// TIA Portal project "LAB5" (V18)

(* hardware
DEVICE "S7-1500/ET200MP station_1"  S7-1500 station
   slot 0: "Rail_0"  Rack  6ES7 590-1***0-0AA0
   slot 1: "PLC_1"  CPU 1511-1 PN  6ES7 511-1AK00-0AB0  V1.8
      slot 3: "CPU display_1"  6ES7591-1AA00-0AA0
      slot 32768: "PROFINET interface_1"  X1
         slot 32769: "Port_1"  X1 P1
         slot 32770: "Port_2"  X1 P2
   slot 2: "CM 1542-5_1"  CM 1542-5  6GK7 542-5DX00-0XE0  V1.0
   slot 3: "DI 16x24VDC HF_1"  DI 16x24VDC HF  6ES7 521-1BH00-0AB0  V2.0
   slot 4: "DQ 16x24VDC/0.5A ST_1"  DQ 16x24VDC/0.5A ST  6ES7 522-1BH00-0AB0  V2.0
   slot 5: "AI 8xU/I/RTD/TC ST_1"  AI 8xU/I/RTD/TC ST  6ES7 531-7KF00-0AB0  V1.0
   slot 6: "AQ 4xU/I ST_1"  AQ 4xU/I ST  6ES7 532-5HD00-0AB0  V1.0
DEVICE "GSD device_1"  GSD.Device
   slot 0: "Rack_0"  Rail
   slot 0: "Slave_1"  6SE640X-1PB00-0AA0  V1.0
DEVICE "HMI_1"  KTP600 Basic color PN
   slot 0: "HMI_1"  KTP600 Basic color PN  6AV6 647-0AD11-3AX0  12.0.0.0
   slot 1: "HMI_RT_1"  KTP600 Basic color PN  6AV6 647-0AD11-3AX0  12.0.0.0
   slot 5: "HMI_1.IE_CP_1"  PROFINET Interface  12.0.0.0
      slot 1: "PROFINET Interface_1"  PROFINET Interface
         slot 1: "Port_1"  Port
DEVICE "PC-System_1"  SIMATIC PC station
   slot 0: "SIMATIC PC station"  Rail  SIMATIC PC-Station  V1.0
      slot 125: "Stationmanager"  Station_Manager  V6.0.4
   slot 1: "HMI_RT_2"  WinCC RT Advanced  6AV2 104-0xxxx-xxxx  16.0.0.0
      slot 33792: "Computer interface"  Host interface
   slot 2: "IE general_1"  IE General  IE_CP  V8.2.0
      slot 1: "PROFINET interface"  IEGeneral.Interface.8.2.0
*)

// ===== PLC "PLC_1"  CPU 1511-1 PN =====

VAR_GLOBAL   // PLC tag table "Default tag table"
   "inicio_variador" AT %M0.0 : Bool;
   "Tag_19" AT %M0.1 : Bool;
   "Tag_20" AT %M0.2 : Bool;
   "Tag_21" AT %M0.3 : Bool;
   "Tag_22" AT %M0.4 : Bool;
   "Tag_23" AT %M0.5 : Bool;
   "Tag_24" AT %M0.6 : Bool;
   "Tag_25" AT %M0.7 : Bool;
   "Tag_26" AT %M1.0 : Bool;
   "Tag_27" AT %M1.1 : Bool;
   "Tag_28" AT %M1.2 : Bool;
   "Tag_29" AT %M1.3 : Bool;
   "Tag_30" AT %M1.4 : Bool;
   "Tag_31" AT %M1.5 : Bool;
   "Tag_32" AT %M1.6 : Bool;
   "Tag_33" AT %M1.7 : Bool;
   "Tag_34" AT %M2.0 : Bool;
   "Tag_1" AT %ID18 : DWord;
   "Palabramando" AT %QW18 : Word;
   "velocidadescribir" AT %QW20 : Int;
   "Tag_2" AT %MW90 : Int;
   "palabraestado" AT %IW26 : Word;
   "parametro" AT %QW10 : Word;
   "indice" AT %QW12 : Word;
   "valorparametro" AT %QD14 : DWord;
   "Tag_4" AT %QW16 : Word;
   "leerparametro" AT %IW18 : Word;
   "paramrecib" AT %MW4 : Word;
   "indicerecib" AT %MW6 : Word;
   "leerindice" AT %IW20 : Word;
   "leervalparametro" AT %ID22 : DWord;
   "valorparamrecib" AT %MD8 : DWord;
   "aux_SP" AT %IW12 : Int;
   "SP" AT %MD16 : Real;
   "Visual_SP" AT %QW22 : Int;
   "aux_Sensor" AT %IW24 : Int;
   "Level_Sensor" AT %MD28 : Real;
   "Visual_Sensor" AT %QW32 : Int;
   "Q_PID" AT %MD36 : Real;
   "Error" AT %MD62 : Real;
   "Start" AT %I0.0 : Bool;
   "Stop" AT %M48.1 : Bool;
   "Emergency" AT %M48.2 : Bool;
   "ON/OFF" AT %M48.3 : Bool;
   "PID" AT %M48.4 : Bool;
   "END" AT %M48.5 : Bool;
   "Reset" AT %M48.6 : Bool;
   "M_Level_CM" AT %MD49 : Real;
   "HMI_SP" AT %MD53 : Real;
   "Q_VFD_Speed" AT %MW58 : Int;
   "Q_Indc_Alarm" AT %Q60.1 : Bool;
   "Q_Indc_Start" AT %Q60.2 : Bool;
   "Q_Indc_Stop" AT %Q60.3 : Bool;
   "Clock1.5Hz" AT %Q60.4 : Bool;
   "Q_Valve" AT %Q60.5 : Bool;
   "M_Limit_Histerisis" AT %QD61 : Real;
   "On_factory" AT %M66.0 : Bool;
   "On_Analogic" AT %M66.1 : Bool;
   "L_Level_Raw" AT %MW67 : Int;
   "L_Level_m" AT %MD70 : Real;
   "SP_%" AT %MD74 : Real;
   "Sensor_%" AT %MD78 : Real;
   "SP_cm" AT %MD82 : Real;
   "Sensor_cm" AT %MD86 : Real;
   "Q_PID_aux" AT %MD92 : Real;
   "M_PID" AT %MD96 : Real;
   "Q_factory" AT %MW120 : Int;
   "Filling" AT %MW102 : Int;
   "Emptying" AT %MW104 : Int;
   "In_Pot" AT %ID30 : Real;
   "In_Sensor" AT %ID34 : Real;
   "Q_PUMP1" AT %QD30 : Real;
   "Q_PUMP2" AT %QD34 : Real;
END_VAR

TYPE "inn"
   STRUCT
      Mandoderecha : Bool;
      Mandoizquierdo : Bool;
      ControldesdePLC : Bool;
      Inversionvalorconsigna : Bool;
      Noutilizado : Bool;
      Potenciometrohaciaarriba : Bool;
      Potenciometrohaciaabajo : Bool;
      "Local/remoto" : Bool;
      "ON/OFF1" : Bool;
      OFF2stopelectrico : Bool;
      OFF3stoprapido : Bool;
      Activarpulsos : Bool;
      Activargeneradorrampa : Bool;
      Generadorrampa : Bool;
      Activarvalorconsigna : Bool;
      Acusedefallo : Bool;
      Velocidadvariador : Int;
   END_STRUCT;
END_TYPE

TYPE "out"
   STRUCT
      Sindesviacionvalreaconsigna : Bool;
      Controlsolicitado : Bool;
      frecuenciasalida : Bool;
      alarma : Bool;
      freno : Bool;
      sobrecarga : Bool;
      giro : Bool;
      sobrecargaconvertidor : Bool;
      listoparaservicio : Bool;
      listoparaarrancar : Bool;
      serviciodesbloqueado : Bool;
      fallo : Bool;
      "comando aus2/off2" : Bool;
      "comandoaus3/off3" : Bool;
      Bloqueodearranque : Bool;
      Alarmas : Bool;
      Velocidadactual : Int;
   END_STRUCT;
END_TYPE

DATA_BLOCK "lect_variador"   // DB1
{ S7_Optimized_Access := 'FALSE' }
VERSION : 0.1
   VAR
      estadovariador : "out";
   END_VAR
BEGIN
END_DATA_BLOCK

DATA_BLOCK "esc_variador"   // DB2
{ S7_Optimized_Access := 'FALSE' }
VERSION : 0.1
   VAR
      esc_variador : "inn";
   END_VAR
BEGIN
END_DATA_BLOCK

DATA_BLOCK "Variator_DB"   // DB3
{ S7_Optimized_Access := 'TRUE' }
VERSION : 0.1
// stored: InstanceOfName Variator
"Variator"
BEGIN
END_DATA_BLOCK

DATA_BLOCK "SETPOINT_DB"   // DB5
{ S7_Optimized_Access := 'TRUE' }
VERSION : 0.1
// stored: InstanceOfName SETPOINT
"SETPOINT"
BEGIN
END_DATA_BLOCK

DATA_BLOCK "SENSOR_DB"   // DB6
{ S7_Optimized_Access := 'TRUE' }
VERSION : 0.1
// stored: InstanceOfName SENSOR
"SENSOR"
BEGIN
END_DATA_BLOCK

DATA_BLOCK "OUT_PID_DB"   // DB7
{ S7_Optimized_Access := 'TRUE' }
VERSION : 0.1
// stored: InstanceOfName OUT_PID
"OUT_PID"
BEGIN
END_DATA_BLOCK

FUNCTION_BLOCK "Variator"   // FB1, LAD
{ S7_Optimized_Access := 'TRUE' }
VERSION : 0.1
BEGIN

REGION Network 1
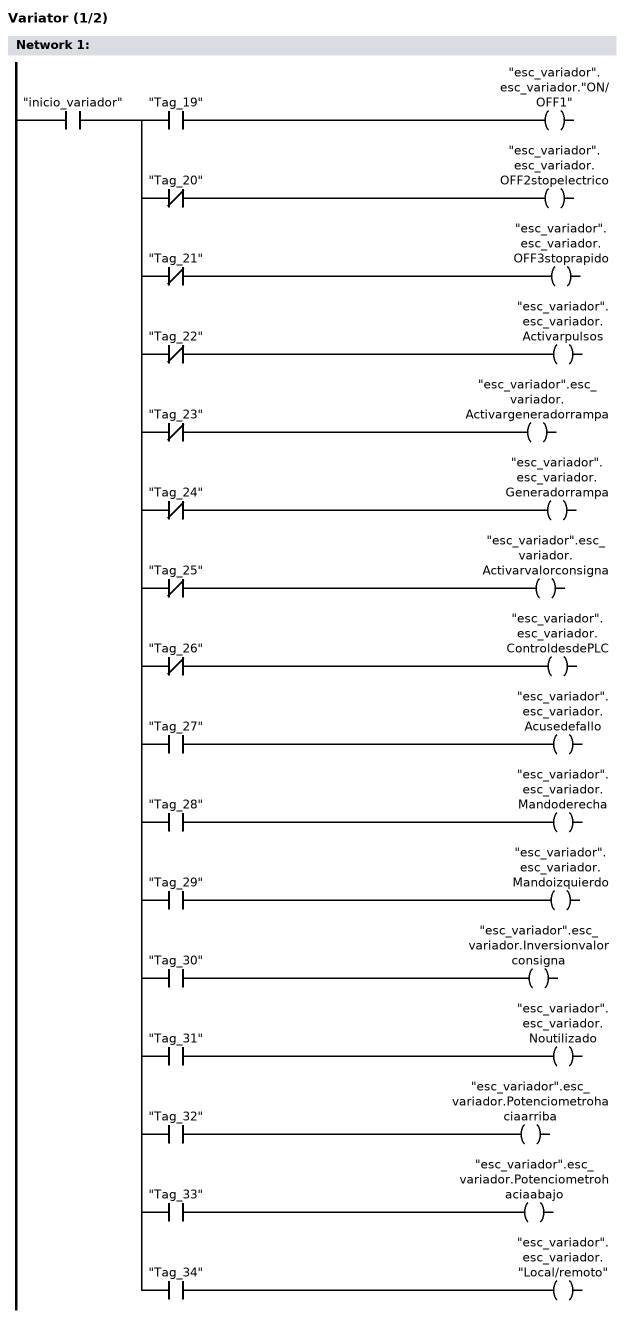
   RUNG wire#powerrail
      Contact( "inicio_variador" )
      wire#w1
      Contact( "Tag_19" )
      Coil( "esc_variador".esc_variador."ON/OFF1" )
   END_RUNG
   RUNG wire#w1
      I_Contact( "Tag_20" )
      Coil( "esc_variador".esc_variador.OFF2stopelectrico )
   END_RUNG
   RUNG wire#w1
      I_Contact( "Tag_21" )
      Coil( "esc_variador".esc_variador.OFF3stoprapido )
   END_RUNG
   RUNG wire#w1
      I_Contact( "Tag_22" )
      Coil( "esc_variador".esc_variador.Activarpulsos )
   END_RUNG
   RUNG wire#w1
      I_Contact( "Tag_23" )
      Coil( "esc_variador".esc_variador.Activargeneradorrampa )
   END_RUNG
   RUNG wire#w1
      I_Contact( "Tag_24" )
      Coil( "esc_variador".esc_variador.Generadorrampa )
   END_RUNG
   RUNG wire#w1
      I_Contact( "Tag_25" )
      Coil( "esc_variador".esc_variador.Activarvalorconsigna )
   END_RUNG
   RUNG wire#w1
      I_Contact( "Tag_26" )
      Coil( "esc_variador".esc_variador.ControldesdePLC )
   END_RUNG
   RUNG wire#w1
      Contact( "Tag_27" )
      Coil( "esc_variador".esc_variador.Acusedefallo )
   END_RUNG
   RUNG wire#w1
      Contact( "Tag_28" )
      Coil( "esc_variador".esc_variador.Mandoderecha )
   END_RUNG
   RUNG wire#w1
      Contact( "Tag_29" )
      Coil( "esc_variador".esc_variador.Mandoizquierdo )
   END_RUNG
   RUNG wire#w1
      Contact( "Tag_30" )
      Coil( "esc_variador".esc_variador.Inversionvalorconsigna )
   END_RUNG
   RUNG wire#w1
      Contact( "Tag_31" )
      Coil( "esc_variador".esc_variador.Noutilizado )
   END_RUNG
   RUNG wire#w1
      Contact( "Tag_32" )
      Coil( "esc_variador".esc_variador.Potenciometrohaciaarriba )
   END_RUNG
   RUNG wire#w1
      Contact( "Tag_33" )
      Coil( "esc_variador".esc_variador.Potenciometrohaciaabajo )
   END_RUNG
   RUNG wire#w1
      Contact( "Tag_34" )
      Coil( "esc_variador".esc_variador."Local/remoto" )
   END_RUNG
   // the same network as SCL:
   "esc_variador".esc_variador."ON/OFF1" := "inicio_variador" AND "Tag_19";
   "esc_variador".esc_variador.OFF2stopelectrico := "inicio_variador" AND NOT "Tag_20";
   "esc_variador".esc_variador.OFF3stoprapido := "inicio_variador" AND NOT "Tag_21";
   "esc_variador".esc_variador.Activarpulsos := "inicio_variador" AND NOT "Tag_22";
   "esc_variador".esc_variador.Activargeneradorrampa := "inicio_variador" AND NOT "Tag_23";
   "esc_variador".esc_variador.Generadorrampa := "inicio_variador" AND NOT "Tag_24";
   "esc_variador".esc_variador.Activarvalorconsigna := "inicio_variador" AND NOT "Tag_25";
   "esc_variador".esc_variador.ControldesdePLC := "inicio_variador" AND NOT "Tag_26";
   "esc_variador".esc_variador.Acusedefallo := "inicio_variador" AND "Tag_27";
   "esc_variador".esc_variador.Mandoderecha := "inicio_variador" AND "Tag_28";
   "esc_variador".esc_variador.Mandoizquierdo := "inicio_variador" AND "Tag_29";
   "esc_variador".esc_variador.Inversionvalorconsigna := "inicio_variador" AND "Tag_30";
   "esc_variador".esc_variador.Noutilizado := "inicio_variador" AND "Tag_31";
   "esc_variador".esc_variador.Potenciometrohaciaarriba := "inicio_variador" AND "Tag_32";
   "esc_variador".esc_variador.Potenciometrohaciaabajo := "inicio_variador" AND "Tag_33";
   "esc_variador".esc_variador."Local/remoto" := "inicio_variador" AND "Tag_34";
END_REGION

REGION Network 2
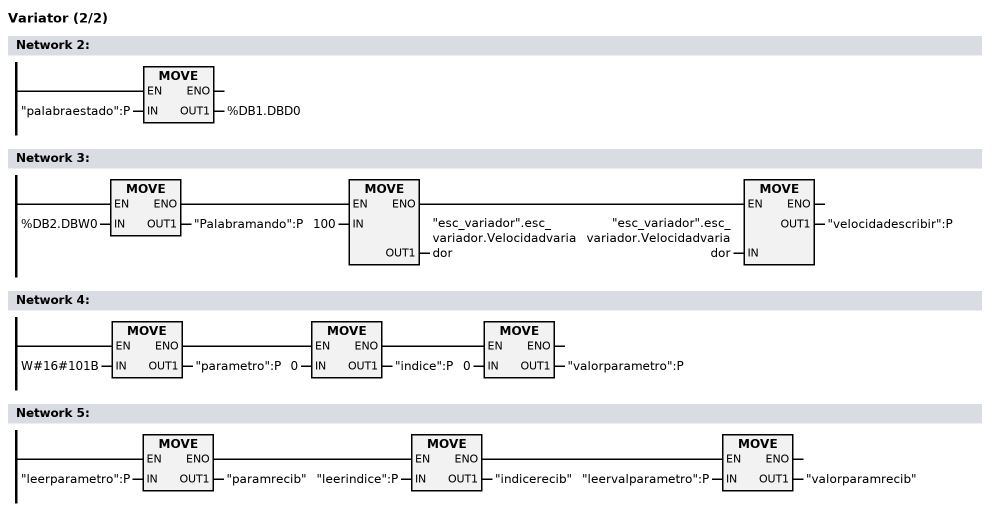
   RUNG wire#powerrail
      Move(in := "palabraestado":P, out1 => %DB1.DBD0)
   END_RUNG
   // the same network as SCL:
   %DB1.DBD0 := "palabraestado":P;
END_REGION

REGION Network 3
   RUNG wire#powerrail
      Move(in := %DB2.DBW0, out1 => "Palabramando":P)
      Move(in := 100, out1 => "esc_variador".esc_variador.Velocidadvariador)
      Move(in := "esc_variador".esc_variador.Velocidadvariador, out1 => "velocidadescribir":P)
   END_RUNG
   // the same network as SCL:
   "Palabramando":P := %DB2.DBW0;
   "esc_variador".esc_variador.Velocidadvariador := 100;
   "velocidadescribir":P := "esc_variador".esc_variador.Velocidadvariador;
END_REGION

REGION Network 4
   RUNG wire#powerrail
      Move(in := W#16#101B, out1 => "parametro":P)
      Move(in := 0, out1 => "indice":P)
      Move(in := 0, out1 => "valorparametro":P)
   END_RUNG
   // the same network as SCL:
   "parametro":P := W#16#101B;
   "indice":P := 0;
   "valorparametro":P := 0;
END_REGION

REGION Network 5
   RUNG wire#powerrail
      Move(in := "leerparametro":P, out1 => "paramrecib")
      Move(in := "leerindice":P, out1 => "indicerecib")
      Move(in := "leervalparametro":P, out1 => "valorparamrecib")
   END_RUNG
   // the same network as SCL:
   "paramrecib" := "leerparametro":P;
   "indicerecib" := "leerindice":P;
   "valorparamrecib" := "leervalparametro":P;
END_REGION
END_FUNCTION_BLOCK

FUNCTION_BLOCK "Program"   // FB2, FBD
{ S7_Optimized_Access := 'TRUE' }
VERSION : 0.1
BEGIN

REGION Network 1: Normalizate and Scale - Factory IO
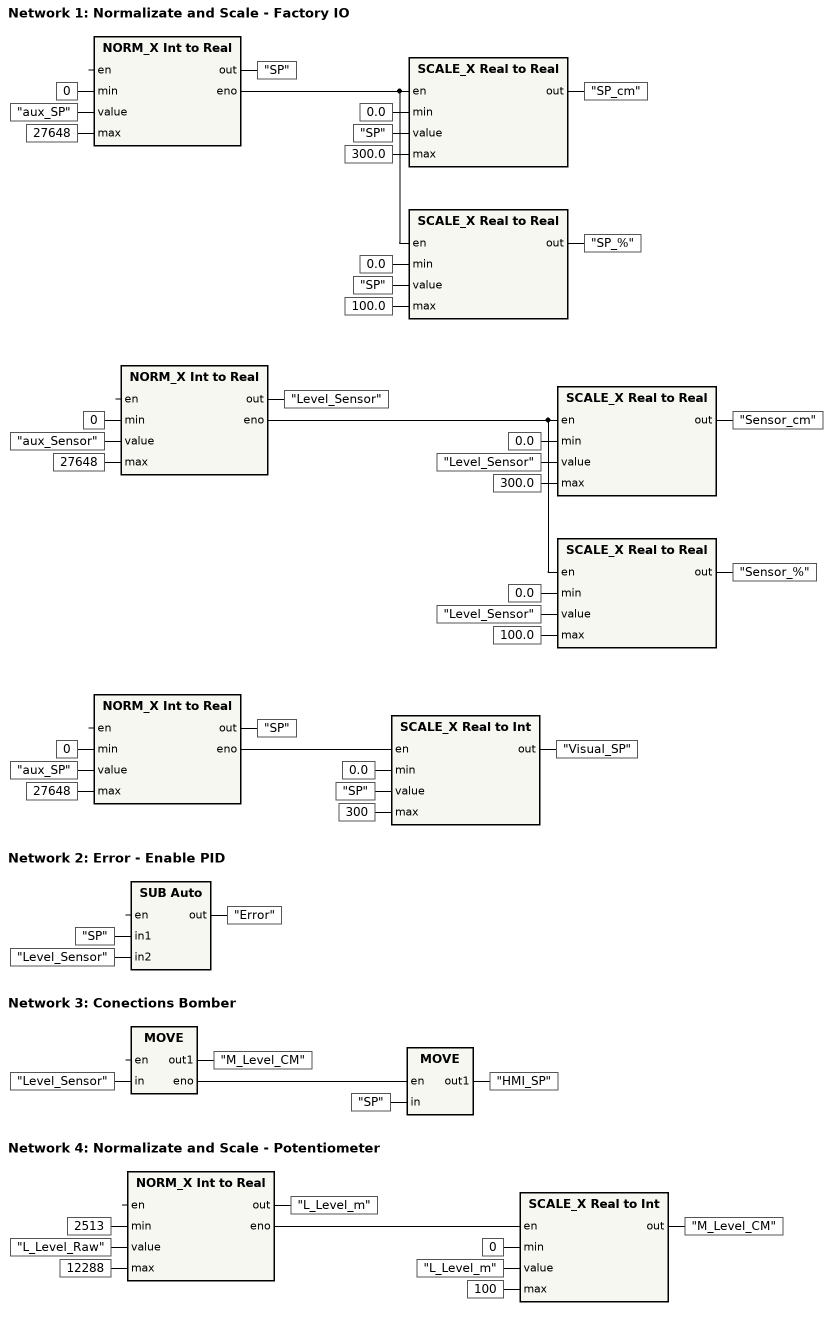
   "SP" := NORM_X(MIN := 0, VALUE := "aux_SP", MAX := 27648);
   "SP_cm" := SCALE_X(MIN := 0.0, VALUE := "SP", MAX := 300.0);
   "SP_%" := SCALE_X(MIN := 0.0, VALUE := "SP", MAX := 100.0);
   "Level_Sensor" := NORM_X(MIN := 0, VALUE := "aux_Sensor", MAX := 27648);
   "Sensor_cm" := SCALE_X(MIN := 0.0, VALUE := "Level_Sensor", MAX := 300.0);
   "Sensor_%" := SCALE_X(MIN := 0.0, VALUE := "Level_Sensor", MAX := 100.0);
   "SP" := NORM_X(MIN := 0, VALUE := "aux_SP", MAX := 27648);
   "Visual_SP" := SCALE_X(MIN := 0.0, VALUE := "SP", MAX := 300);
END_REGION

REGION Network 2: Error - Enable PID
   "Error" := "SP" - "Level_Sensor";
END_REGION

REGION Network 3: Conections Bomber
   "M_Level_CM" := "Level_Sensor";
   "HMI_SP" := "SP";
END_REGION

REGION Network 4: Normalizate and Scale - Potentiometer
   "L_Level_m" := NORM_X(MIN := 2513, VALUE := "L_Level_Raw", MAX := 12288);
   "M_Level_CM" := SCALE_X(MIN := 0, VALUE := "L_Level_m", MAX := 100);
END_REGION

REGION Network 5
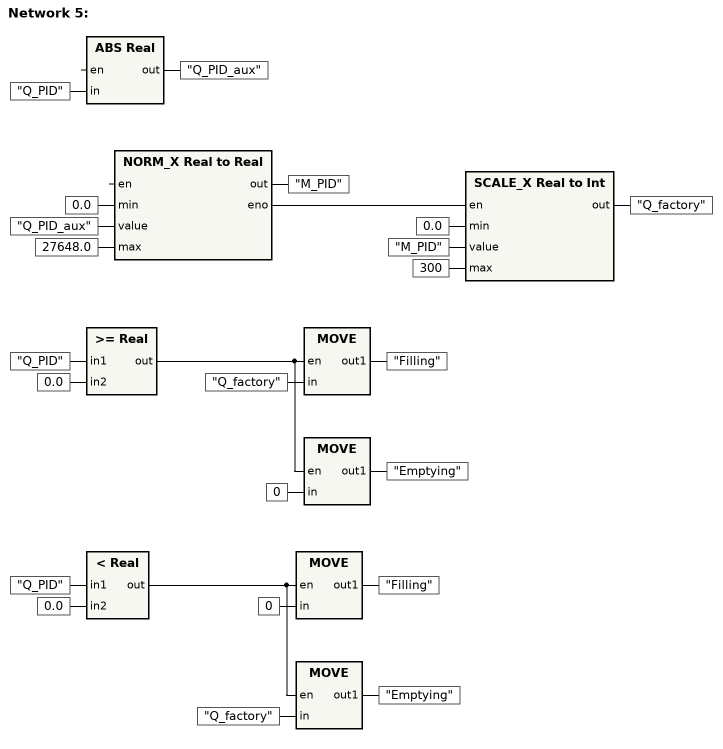
   "Q_PID_aux" := ABS("Q_PID");
   "M_PID" := NORM_X(MIN := 0.0, VALUE := "Q_PID_aux", MAX := 27648.0);
   "Q_factory" := SCALE_X(MIN := 0.0, VALUE := "M_PID", MAX := 300);
   IF "Q_PID" >= 0.0 THEN
       "Filling" := "Q_factory";
       "Emptying" := 0;
   END_IF;
   IF "Q_PID" < 0.0 THEN
       "Filling" := 0;
       "Emptying" := "Q_factory";
   END_IF;
END_REGION
END_FUNCTION_BLOCK

FUNCTION_BLOCK "SETPOINT"   // FB4, FBD
{ S7_Optimized_Access := 'TRUE' }
VERSION : 0.1
   VAR_INPUT
      InAnalog : Int;
   END_VAR
   VAR_OUTPUT
      "SP(cm)" : Real;
      "SP(%)" : Real;
   END_VAR
   VAR
      aux : Real;
   END_VAR
BEGIN

REGION Network 1
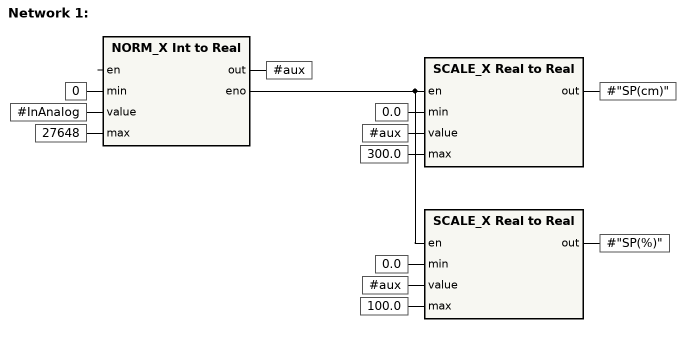
   #aux := NORM_X(MIN := 0, VALUE := #InAnalog, MAX := 27648);
   #"SP(cm)" := SCALE_X(MIN := 0.0, VALUE := #aux, MAX := 300.0);
   #"SP(%)" := SCALE_X(MIN := 0.0, VALUE := #aux, MAX := 100.0);
END_REGION
END_FUNCTION_BLOCK

FUNCTION_BLOCK "SENSOR"   // FB5, FBD
{ S7_Optimized_Access := 'TRUE' }
VERSION : 0.1
   VAR_INPUT
      InAnalog : Int;
   END_VAR
   VAR_OUTPUT
      "Level(cm)" : Real;
      "Level(%)" : Real;
   END_VAR
   VAR
      aux : Real;
   END_VAR
BEGIN

REGION Network 1
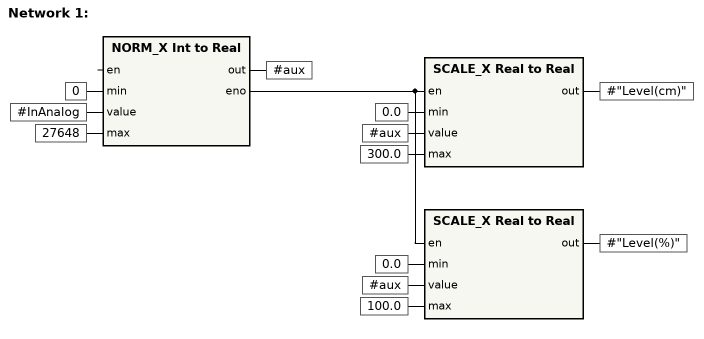
   #aux := NORM_X(MIN := 0, VALUE := #InAnalog, MAX := 27648);
   #"Level(cm)" := SCALE_X(MIN := 0.0, VALUE := #aux, MAX := 300.0);
   #"Level(%)" := SCALE_X(MIN := 0.0, VALUE := #aux, MAX := 100.0);
END_REGION
END_FUNCTION_BLOCK

FUNCTION_BLOCK "OUT_PID"   // FB6, FBD
{ S7_Optimized_Access := 'TRUE' }
VERSION : 0.1
   VAR_INPUT
      Q_PID_M : Real;
   END_VAR
   VAR_OUTPUT
      Pump1 : Int;
      Pump2 : Int;
   END_VAR
   VAR
      aux : Real;
      aux1 : Real;
      Q_Analog : Int;
   END_VAR
BEGIN

REGION Network 1
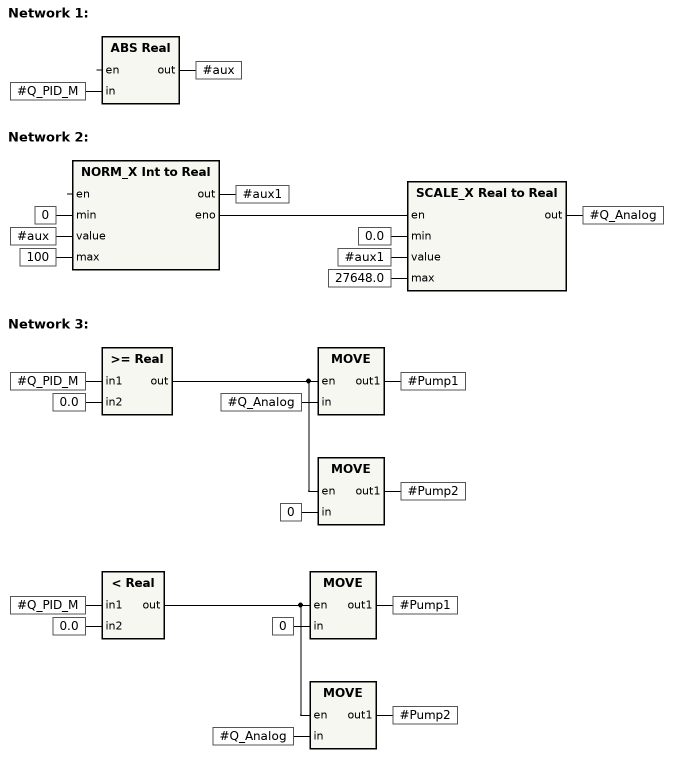
   #aux := ABS(#Q_PID_M);
END_REGION

REGION Network 2
   #aux1 := NORM_X(MIN := 0, VALUE := #aux, MAX := 100);
   #Q_Analog := SCALE_X(MIN := 0.0, VALUE := #aux1, MAX := 27648.0);
END_REGION

REGION Network 3
   IF #Q_PID_M >= 0.0 THEN
       #Pump1 := #Q_Analog;
       #Pump2 := 0;
   END_IF;
   IF #Q_PID_M < 0.0 THEN
       #Pump1 := 0;
       #Pump2 := #Q_Analog;
   END_IF;
END_REGION
END_FUNCTION_BLOCK

ORGANIZATION_BLOCK "Main"   // OB1, LAD, ProgramCycle
TITLE = "Main Program Sweep (Cycle)"
{ S7_Optimized_Access := 'TRUE' }
VERSION : 0.1
   VAR_INPUT
      Initial_Call : Bool;   // Initial call of this OB
      Remanence : Bool;   // =True, if remanent data are available
   END_VAR
   VAR_TEMP
      l : Bool;
      l1 : DWord;
   END_VAR
BEGIN

REGION Network 1
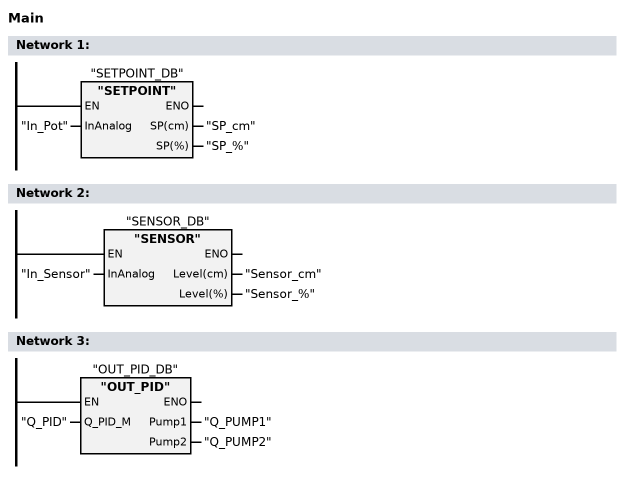
   RUNG wire#powerrail
      "SETPOINT_DB"(InAnalog := "In_Pot", "SP(cm)" => "SP_cm", "SP(%)" => "SP_%")
   END_RUNG
   // the same network as SCL:
   "SETPOINT_DB"(InAnalog := "In_Pot", "SP(cm)" => "SP_cm", "SP(%)" => "SP_%");   // "SETPOINT"
END_REGION

REGION Network 2
   RUNG wire#powerrail
      "SENSOR_DB"(InAnalog := "In_Sensor", "Level(cm)" => "Sensor_cm", "Level(%)" => "Sensor_%")
   END_RUNG
   // the same network as SCL:
   "SENSOR_DB"(InAnalog := "In_Sensor", "Level(cm)" => "Sensor_cm", "Level(%)" => "Sensor_%");   // "SENSOR"
END_REGION

REGION Network 3
   RUNG wire#powerrail
      "OUT_PID_DB"(Q_PID_M := "Q_PID", Pump1 => "Q_PUMP1", Pump2 => "Q_PUMP2")
   END_RUNG
   // the same network as SCL:
   "OUT_PID_DB"(Q_PID_M := "Q_PID", Pump1 => "Q_PUMP1", Pump2 => "Q_PUMP2");   // "OUT_PID"
END_REGION
END_ORGANIZATION_BLOCK

ORGANIZATION_BLOCK "Control"   // OB30, FBD, CyclicInterrupt
{ S7_Optimized_Access := 'TRUE' }
VERSION : 0.1
   VAR_INPUT
      Initial_Call : Bool;   // Initial call of this OB
      Event_Count : Int;   // Events discarded
   END_VAR
BEGIN

REGION Network 1: PID1
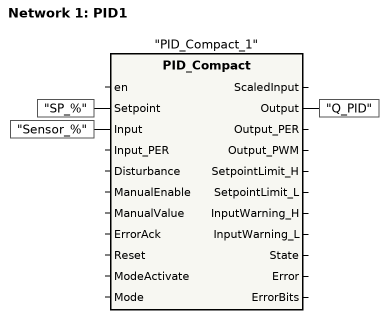
   "PID_Compact_1"(Setpoint := "SP_%", Input := "Sensor_%", Output => "Q_PID");   // PID_Compact
END_REGION
END_ORGANIZATION_BLOCK

(* ===== HMI "HMI_RT_1" =====
system functions are stored by id; their names below are inferred from use
connection "HMI_Connection_3": ETHERNET, SMART_S7_1500_OMS

HMI tags "Default tag table"
   "Inicio" : Bool = PLC Start AT %I0.0, 1 s
   "Arranqu" : Bool = PLC ArranqueFlag AT %M12.6, 1 s
   "Sto" : Bool = PLC Stop AT %M48.1, 1 s
   "Stop_E" : Bool = PLC Stop_EM AT %M12.1, 1 s
   "Nive" : Int = PLC Nivel AT %MW14, 1 s
   "Referenci" : Int = PLC Referencia AT %MW16, 1 s
   "RPM_Actua" : Int = PLC RPM_Actual AT %MW48, 1 s
   "LEH_HMI" : Bool = PLC LEH AT %M12.2, 1 s
   "LEL_HMI" : Bool = PLC LEL AT %M12.3, 1 s
   "Bomb" : Bool = PLC Bomba AT %M12.4, 1 s
   "bomba1" : Bool = PLC Bomba AT %M12.4, 1 s

screen "Root screen" 320x240, template "Template_1"
   GraphicView "Graphic view_8" at 127,163 size 57x37; Picture "Graphic_13"
   GraphicView "Graphic view_2" at 36,49 size 20x17; Picture "Graphic_2"
      Visibility <- "Sto"
   GraphicView "Graphic view_1" at 6,49 size 20x17; Picture "Graphic_1"
      Visibility <- "Arranqu"
   GraphicView "Graphic view_7" at 5,68 size 71x109; Picture "Graphic_7"
   GraphicView "Graphic view_4" at 76,3 size 155x164; Picture "Graphic_4"
   Button "Button_2" at 12,109 size 60x24; TextOff 'Stop'
      on Press: InvertBit("Sto")
   Switch "Pushbutton_Emergency" at 26,136 size 29x28; CaptionText 'Switch'; TextOff '0'; TextOn '1'; PictureOff "Pushbutton_Emergency_Off_256c"; PictureOn "Pushbutton_Emergency_On_256c"
      on Change: InvertBit("Stop_E")
      ProcessValue <- "Stop_E"
   GraphicView "Graphic view_3" at 87,192 size 56x41; Picture "Graphic_3"
      Visibility <- "Bomb"
   Bar "Bar_1" at 99,37 size 120x98; MinimumValue 0; MaximumValue 300
      ProcessValue <- "Nive"
      Visibility <- "Nive"
   GraphicView "Graphic view_5" at 234,36 size 14x50; Picture "Graphic_5"
      Visibility <- "LEH_HMI"
   Button "Button_3" at 253,80 size 59x21; TextOff '100'
      on Press: SetTag("Referenci", 100)
   IOField "I/O field_1" at 192,184 size 77x21; FormatPattern s99999
      ProcessValue <- "Referenci"
   IOField "I/O field_2" at 6,204 size 74x24; FormatPattern s99999
      ProcessValue <- "RPM_Actua"
   TrendView "Trend view_1" at 350,109 size 203x197
   TextField "Text field_1" at 248,43 size 69x32; Text 'Referencia Rápida'
   Button "Button_4" at 253,101 size 59x19; TextOff '80'
      on Press: SetTag("Referenci", 80)
   Button "Button_5" at 253,120 size 59x19; TextOff '60'
      on Press: SetTag("Referenci", 60)
   Button "Button_6" at 253,139 size 59x15; TextOff '40'
      on Press: SetTag("Referenci", 40)
   Button "Button_7" at 253,153 size 59x17; TextOff '20'
      on Press: SetTag("Referenci", 20)
   Button "Button_8" at 253,170 size 59x14; TextOff '0'
      on Press: SetTag("Referenci", 0)
   TextField "Text field_7" at 19,179 size 42x23; Text 'RPM'
   GraphicView "Graphic view_9" at 139,198 size 35x30; Picture "Graphic_9"
   Button "Button_9" at 241,206 size 68x30; TextOff 'Grafica'
      on Click: ActivateScreen("Screen_1", 0)
   Button "Button_1" at 14,79 size 53x27; TextOff 'star'
      on Press: InvertBit("Inicio")
   Button "Button_10" at 239,8 size 74x26; TextOff 'Punto2'
      on Click: ActivateScreen("Screen_2", 0)

screen "Screen_1" 320x240
   TrendView "Trend view_1" at 30,54 size 258x174
   Button "Button_1" at 105,13 size 96x32; TextOff 'Text'
      on Click: ActivateScreen("Root screen", 0)

screen "Screen_2" 320x240
   Button "Button_1" at 263,5 size 50x27; TextOff 'punto1'
      on Click: ActivateScreen("Root screen", 0)
   GraphicView "Graphic view_1" at 107,47 size 213x192; Picture "Graphic_14"
   TextField "Text field_1" at 158,136 size 10x13; Text 'A'
   TextField "Text field_2" at 218,68 size 10x13; Text 'B'
   TextField "Text field_3" at 278,0 size 10x13; Text 'A'
   TextField "Text field_4" at 282,130 size 10x13; Text 'C'
   TextField "Text field_5" at 158,163 size 10x13; Text 'D'
   TextField "Text field_6" at 219,210 size 10x13; Text 'E'
   TextField "Text field_7" at 119,6 size 48x13; Text 'PUNTO 2'
   GraphicView "Graphic view_7" at 16,56 size 71x109; Picture "Graphic_7"

Template "Template_1" 320x240
   Button "Exit" at 714,429 size 71x50; TextOn 'Exit'; TextOff 'Exit'; PictureOn "ExitRuntime_KTP700_Basic_PN_TR"; PictureOff "ExitRuntime_KTP700_Basic_PN_TR"
      on Release: StopRuntime(0)
   Button "Template_Button" at 614,429 size 71x50; TextOff 'Text'
   Button "Template_Button_1" at 514,429 size 71x50; TextOff 'Text'
   Button "Template_Button_2" at 414,429 size 71x50; TextOff 'Text'
   Button "Template_Button_3" at 314,429 size 71x50; TextOff 'Text'
   Button "Template_Button_4" at 214,429 size 71x50; TextOff 'Text'
   Button "Alarms" at 114,429 size 71x50; TextOn 'Alarms'; TextOff 'Alarms'; PictureOn "AlarmDisplay_KTP700_Basic_PN_TR"; PictureOff "AlarmDisplay_KTP700_Basic_PN_TR"
      on Release: function_ef3f5d25("Alarm window_Unacknowledged", -1)
   Button "Start screen" at 14,429 size 71x50; TextOn 'Start screen'; TextOff 'Start screen'; PictureOn "NavigateHome_KTP700_Basic_PN_TR"; PictureOff "NavigateHome_KTP700_Basic_PN_TR"
      on Release: ActivateScreen("Root screen", 0)
   DateTimeField "HmiScreenItemData" at 695,25 size 105x25
   DateTimeField "HmiScreenItemData_1" at 695,0 size 105x25
   GraphicView "Logo" at 0,0 size 91x51; Picture "Logo of HMI_1"
*)

(* ===== HMI "HMI_RT_2" =====
system functions are stored by id; their names below are inferred from use
connection "HMI_Connection_2": ETHERNET, S7_1500_OMS

HMI tags "Default tag table"
   "Arranqu1" : Bool = PLC Tag_27 AT %M1.1, 1 s
   "Inicio1" : Bool = PLC Start AT %I0.0, 1 s
   "Nive1" : Int = PLC Nivel AT %MW14, 1 s
   "Referenci1" : Int = PLC Referencia AT %MW16, 1 s
   "Sto1" : Bool = PLC Stop AT %M48.1, 1 s
   "Stop_E1" : Bool = PLC Stop_EM AT %M12.1, 1 s
   "RPM_Actua1" : Int = PLC RPM_Actual AT %MW48, 1 s
   "LEH_HMI1" : Bool = PLC LEH AT %M12.2, 1 s
   "LEL_HMI1" : Bool = PLC LEL AT %M12.3, 1 s
   "Bomb1" : Bool = PLC Tag_32 AT %M1.6, 1 s
   "pid1" : Bool = PLC PID AT %M48.4, 1 s
   "onoff1" : Bool = PLC onoff AT %M22.1, 1 s
   "punto1.1" : Bool = PLC punto1 AT %M50.0, 1 s
   "punto2.2" : Bool = PLC punto2 AT %M50.1, 1 s
   "actuadorb" : Bool = PLC actuadorB AT %M52.0, 1 s
   "actuadorc1" : Bool = PLC actuadorc1 AT %M52.1, 1 s
   "actuadorc2" : Bool = PLC actuadorc2 AT %M52.2, 1 s
   "actuadore" : Bool = PLC actuadore AT %M52.3, 1 s
   "derecha" : Bool = PLC servoderecha AT %M52.5, 1 s
   "izquierda" : Bool = PLC servoizquierda AT %M52.4, 1 s
   "peso1" : Int = PLC peso AT %MW58, 1 s
   "cambionivel" : Bool = PLC cambiodenivel AT %M30.0, 1 s

screen "Screen_1" 1024x768
   GraphicView "Graphic view_3" at 197,324 size 129x73; Picture "Graphic_3"
      Visibility <- "Bomb1"
   GraphicView "Graphic view_8" at 322,345 size 34x34; Picture "Graphic_9"
   GraphicView "Graphic view_10" at 298,311 size 80x37; Picture "Graphic_13"
   GraphicView "Graphic view_4" at 248,102 size 187x217; Picture "Graphic_4"
   Button "Button_1" at 78,173 size 66x17; TextOff 'Start'
      on Press: InvertBit("Inicio1")
      Visibility <- "Inicio1"
   Button "Button_2" at 66,135 size 96x32; TextOff 'Stop'
      on Press: InvertBit("Sto1")
   Switch "Pushbutton_Emergency" at 82,233 size 64x62; CaptionText 'Switch'; TextOff '0'; TextOn '1'; PictureOff "Pushbutton_Emergency_Off_256c"; PictureOn "Pushbutton_Emergency_On_256c"
      on Change: InvertBit("Stop_E1")
   Bar "Bar_1" at 280,161 size 115x120; MinimumValue 0; MaximumValue 100
      Visibility <- "Nive1"
      ProcessValue <- "Nive1"
   GraphicView "Graphic view_5" at 404,98 size 14x50; Picture "Graphic_5"
      Visibility <- "LEH_HMI1"
   GraphicView "Graphic view_6" at 199,323 size 27x29; Picture "Graphic_6"
      Visibility <- "LEL_HMI1"
   Button "Button_3" at 435,126 size 84x22; TextOff '100'
      on Press: SetTag("Referenci1", 100)
   IOField "I/O field_1" at 214,401 size 96x32; FormatPattern s99999
      ProcessValue <- "Referenci1"
   IOField "I/O field_2" at 212,352 size 96x32; FormatPattern s99999
      ProcessValue <- "RPM_Actua1"
   TrendView "Trend view_1" at 540,88 size 379x264
   TextField "Text field_1" at 431,83 size 93x42; Text 'Referencia'
   TextField "Text field_2" at 210,436 size 93x61; Text 'Referencia por Texto'
   TextField "Text field_3" at 31,21 size 635x40; Text 'Guía 5 Supervisión Julian , Juanita, Daniel'
   Button "Button_4" at 435,149 size 84x22; TextOff '80'
      on Press: SetTag("Referenci1", 80)
   Button "Button_5" at 435,173 size 84x22; TextOff '60'
      on Press: SetTag("Referenci1", 60)
   Button "Button_6" at 435,197 size 84x22; TextOff '40'
      on Press: SetTag("Referenci1", 40)
   Button "Button_7" at 435,221 size 84x22; TextOff '20'
      on Press: SetTag("Referenci1", 20)
   Button "Button_8" at 435,245 size 84x22; TextOff '0'
      on Press: SetTag("Referenci1", 0)
   TextField "Text field_6" at 47,295 size 125x18; Text 'Paro de Emergencia'
   TextField "Text field_7" at 238,325 size 42x23; Text 'RPM'
   Button "Button_9" at 73,198 size 76x27; TextOff 'PLAY'
      on Press: InvertBit("Inicio1")
   Button "Button_10" at 800,48 size 96x32; TextOff 'PID'
      on Press: InvertBit("pid1")
      Appearance <- "pid1"
   Button "Button_11" at 810,365 size 96x32; TextOff 'ON/OFF'
      on Press: InvertBit("onoff1")
      Appearance <- "onoff1"
   Button "Button_12" at 21,83 size 171x32; TextOff 'Activar punto1'
      on Click: InvertBit("punto1.1")
      Appearance <- "punto1.1"
   Button "Button_13" at 21,323 size 172x49; TextOff 'Interfaz Punto 2'
      on Click: ActivateScreen("Screen_2", 0)
   Button "Button_14" at 88,501 size 355x108; TextOff 'Modo de lectura de nivel potenciometro'
      on Click: InvertBit("cambionivel")
      Appearance <- "cambionivel"

screen "Screen_2" 1024x768
   Button "Button_1" at 23,325 size 152x37; TextOff 'Interfaz Punto 1'
      on Click: ActivateScreen("Screen_1", 0)
   GraphicView "Graphic view_7" at 17,104 size 153x197; Picture "Graphic_7"
   Switch "Pushbutton_Emergency" at 64,215 size 64x62; CaptionText 'Switch'; TextOff '0'; TextOn '1'; PictureOff "Pushbutton_Emergency_Off_256c"; PictureOn "Pushbutton_Emergency_On_256c"
      on Change: InvertBit("Stop_E1")
   TextField "Text field_6" at 36,275 size 125x18; Text 'Paro de Emergencia'
   Button "Button_2" at 26,31 size 146x45; TextOff 'Activar Punto 2'
      on Click: InvertBit("punto2.2")
      Appearance <- "punto2.2"
   GraphicView "Graphic view_1" at 202,31 size 614x489; Picture "Graphic_14"
      Appearance <- "actuadore"
   Rectangle "Rectangle_1" at 379,242 size 76x29
      Appearance <- "actuadorc1"
   Rectangle "Rectangle_2" at 515,127 size 29x71
      Appearance <- "actuadorb"
   Rectangle "Rectangle_3" at 609,244 size 66x23
      Appearance <- "actuadorc2"
   Rectangle "Rectangle_4" at 400,332 size 65x26
      Appearance <- "izquierda"
   TextField "Text field_1" at 355,253 size 15x22; Text 'A'
   TextField "Text field_2" at 529,104 size 15x22; Text 'B'
   TextField "Text field_3" at 681,253 size 15x22; Text 'C'
   TextField "Text field_4" at 375,338 size 16x22; Text 'D'
   TextField "Text field_5" at 524,460 size 14x22; Text 'E'
   Rectangle "Rectangle_6" at 592,334 size 65x26
      Appearance <- "derecha"
   TextField "Text field_7" at 665,338 size 16x22; Text 'D'
   IOField "I/O field_1" at 56,378 size 96x32; FormatPattern s99999
      ProcessValue <- "peso1"
   TextField "Text field_8" at 78,410 size 46x22; Text 'PESO'
*)